PROGRAM POU
VAR
END_VAR

// NETWORK 1

END_PROGRAM

(* stored: Version 1.1.0.1, ProductVersion 3.1.4024.12
   POU POU: Id {492deb71-3555-4e85-ae5f-ef30d01725d1}, SpecialFunc None *)
